PROGRAM MAIN_GENERAR_POLS
VAR
	VARIABLE_A_PULSAR: BOOL;
	GENERA_POLS: BOOL;
END_VAR

VARIABLE_A_PULSAR := GENERAR_POLS(Pols_ON:= GENERA_POLS, Temps_pols:= T#2000ms);

END_PROGRAM

(* stored: Version 1.1.0.1, ProductVersion 3.1.4024.12
   POU MAIN_GENERAR_POLS: Id {f3990073-cdee-4b91-839f-e2718e4d2efa}, SpecialFunc None *)
